(* IEC 61131-3 sources: ATCMcontrol_Engineering/src/Target/ATHW119/Libs/ATCM_Utility, 30 files *)

(* ---- BYTE_SWAP_DWORD.st ---- *)
(*[[
    UserURL= "ATCMfile:BYTE_SWAP_DWORD.htm"
]]*)

(* swaps from big to little endian byte order and vice versa *)

FUNCTION BYTE_SWAP_DWORD : DWORD
VAR_INPUT
    VALUE : DWORD;
END_VAR

inline { STDLIB ( byte_swap_dword ) }

END_FUNCTION

(* ---- BYTE_SWAP_WORD.st ---- *)
(*[[
    UserURL= "ATCMfile:BYTE_SWAP_WORD.htm"
]]*)

(* swaps from big to little endian byte order and vice versa *)

FUNCTION BYTE_SWAP_WORD : WORD
VAR_INPUT
    VALUE : WORD;
END_VAR

inline { STDLIB ( byte_swap_word ) }

END_FUNCTION

(* ---- COPY_BOOL_FROM_BYTE_ARRAY.st ---- *)
(*[[
    UserURL= "ATCMfile:COPY_BOOL_FROM_BYTE_ARRAY.htm"
]]*)

(* returns a value copied from the byte array at the position POS *)

FUNCTION COPY_BOOL_FROM_BYTE_ARRAY : BOOL
VAR_IN_OUT
    POS : DINT;
    BYTES : ARRAY OF BYTE;
END_VAR

inline { STDLIB ( copy_bool_from_byte_array ) }

END_FUNCTION

(* ---- COPY_BOOL_TO_BYTE_ARRAY.st ---- *)
(*[[
    UserURL= "ATCMfile:COPY_BOOL_TO_BYTE_ARRAY.htm"
]]*)

(* copies the value VALUE to the byte array at the position POS *)

FUNCTION COPY_BOOL_TO_BYTE_ARRAY
VAR_INPUT
    VALUE : BOOL;
END_VAR
VAR_IN_OUT
    POS : DINT;
    BYTES : ARRAY OF BYTE;
END_VAR

inline { STDLIB ( copy_bool_to_byte_array ) }

END_FUNCTION

(* ---- COPY_BYTE_FROM_BYTE_ARRAY.st ---- *)
(*[[
    UserURL= "ATCMfile:COPY_BYTE_FROM_BYTE_ARRAY.htm"
]]*)

(* returns a value copied from the byte array BYTES at the position POS *)

FUNCTION COPY_BYTE_FROM_BYTE_ARRAY : BYTE
VAR_IN_OUT
    POS : DINT;
    BYTES : ARRAY OF BYTE;
END_VAR

inline { STDLIB ( copy_byte_from_byte_array ) }

END_FUNCTION

(* ---- COPY_BYTE_TO_BYTE_ARRAY.st ---- *)
(*[[
    UserURL= "ATCMfile:COPY_BYTE_TO_BYTE_ARRAY.htm"
]]*)

(* copies the value VALUE to the byte array BYTES at the position POS *)

FUNCTION COPY_BYTE_TO_BYTE_ARRAY
VAR_INPUT
    VALUE : BYTE;
END_VAR
VAR_IN_OUT
    POS : DINT;
    BYTES : ARRAY OF BYTE;
END_VAR

inline { STDLIB ( copy_byte_to_byte_array ) }

END_FUNCTION

(* ---- COPY_DINT_FROM_BYTE_ARRAY.st ---- *)
(*[[
    UserURL= "ATCMfile:COPY_DINT_FROM_BYTE_ARRAY.htm"
]]*)

(* returns a value copied from the byte array BYTES at the position POS *)

FUNCTION COPY_DINT_FROM_BYTE_ARRAY : DINT
VAR_IN_OUT
    POS : DINT;
    BYTES : ARRAY OF BYTE;
END_VAR

inline { STDLIB ( copy_dint_from_byte_array ) }

END_FUNCTION

(* ---- COPY_DINT_TO_BYTE_ARRAY.st ---- *)
(*[[
    UserURL= "ATCMfile:COPY_DINT_TO_BYTE_ARRAY.htm"
]]*)

(* copies the value VALUE to the byte array BYTES at the position POS *)

FUNCTION COPY_DINT_TO_BYTE_ARRAY
VAR_INPUT
    VALUE : DINT;
END_VAR
VAR_IN_OUT
    POS : DINT;
    BYTES : ARRAY OF BYTE;
END_VAR

inline { STDLIB ( copy_dint_to_byte_array ) }

END_FUNCTION

(* ---- COPY_DWORD_FROM_BYTE_ARRAY.st ---- *)
(*[[
    UserURL= "ATCMfile:COPY_DWORD_FROM_BYTE_ARRAY.htm"
]]*)

(* returns a value copied from the byte array at the position POS *)

FUNCTION COPY_DWORD_FROM_BYTE_ARRAY : DWORD
VAR_IN_OUT
    POS : DINT;
    BYTES : ARRAY OF BYTE;
END_VAR

inline { STDLIB ( copy_dword_from_byte_array ) }

END_FUNCTION

(* ---- COPY_DWORD_TO_BYTE_ARRAY.st ---- *)
(*[[
    UserURL= "ATCMfile:COPY_DWORD_TO_BYTE_ARRAY.htm"
]]*)

(* copies the value VALUE to the byte array at the position POS *)

FUNCTION COPY_DWORD_TO_BYTE_ARRAY
VAR_INPUT
    VALUE : DWORD;
END_VAR
VAR_IN_OUT
    POS : DINT;
    BYTES : ARRAY OF BYTE;
END_VAR

inline { STDLIB ( copy_dword_to_byte_array ) }

END_FUNCTION

(* ---- COPY_INT_FROM_BYTE_ARRAY.st ---- *)
(*[[
    UserURL= "ATCMfile:COPY_INT_FROM_BYTE_ARRAY.htm"
]]*)

(* returns a value copied from the byte string BSTR at the position POS *)

FUNCTION COPY_INT_FROM_BYTE_ARRAY : INT
VAR_IN_OUT
    POS : DINT;
    BYTES : ARRAY OF BYTE;
END_VAR

inline { STDLIB ( copy_int_from_byte_array ) }

END_FUNCTION

(* ---- COPY_INT_TO_BYTE_ARRAY.st ---- *)
(*[[
    UserURL= "ATCMfile:COPY_INT_TO_BYTE_ARRAY.htm"
]]*)

(* copies the value VALUE to the byte array BYTES at the position POS *)
FUNCTION COPY_INT_TO_BYTE_ARRAY
VAR_INPUT
    VALUE : INT;
END_VAR
VAR_IN_OUT
    POS : DINT;
    BYTES : ARRAY OF BYTE;
END_VAR

inline { STDLIB ( copy_int_to_byte_array ) }

END_FUNCTION

(* ---- COPY_LREAL_FROM_BYTE_ARRAY.st ---- *)
(*[[
    UserURL= "ATCMfile:COPY_LREAL_FROM_BYTE_ARRAY.htm"
]]*)

(* returns a value copied from the byte string BSTR at the position POS *)

FUNCTION COPY_LREAL_FROM_BYTE_ARRAY : LREAL
VAR_IN_OUT
    POS : DINT;
    BYTES : ARRAY OF BYTE;
END_VAR

inline { STDLIB ( copy_lreal_from_byte_array ) }

END_FUNCTION

(* ---- COPY_LREAL_TO_BYTE_ARRAY.st ---- *)
(*[[
    UserURL= "ATCMfile:COPY_LREAL_TO_BYTE_ARRAY.htm"
]]*)

(* copies the value VALUE to the byte string BSTR at the position POS *)

FUNCTION COPY_LREAL_TO_BYTE_ARRAY
VAR_INPUT
    VALUE : LREAL;
END_VAR
VAR_IN_OUT
    POS : DINT;
    BYTES : ARRAY OF BYTE;
END_VAR

inline { STDLIB ( copy_lreal_to_byte_array ) }

END_FUNCTION

(* ---- COPY_LWORD_FROM_BYTE_ARRAY.st ---- *)
(*[[
    UserURL= "ATCMfile:COPY_LWORD_FROM_BYTE_ARRAY.htm"
]]*)

(* returns a value copied from the byte string BSTR at the position POS *)

FUNCTION COPY_LWORD_FROM_BYTE_ARRAY : LWORD
VAR_IN_OUT
    POS : DINT;
    BYTES : ARRAY OF BYTE;
END_VAR

inline { STDLIB ( copy_lword_from_byte_array ) }

END_FUNCTION

(* ---- COPY_LWORD_TO_BYTE_ARRAY.st ---- *)
(*[[
    UserURL= "ATCMfile:COPY_LWORD_TO_BYTE_ARRAY.htm"
]]*)

(* copies the value VALUE to the byte string BSTR at the position POS *)

FUNCTION COPY_LWORD_TO_BYTE_ARRAY
VAR_INPUT
    VALUE : LWORD;
END_VAR
VAR_IN_OUT
    POS : DINT;
    BYTES : ARRAY OF BYTE;
END_VAR

inline { STDLIB ( copy_lword_to_byte_array ) }

END_FUNCTION

(* ---- COPY_REAL_FROM_BYTE_ARRAY.st ---- *)
(*[[
    UserURL= "ATCMfile:COPY_LREAL_FROM_BYTE_ARRAY.htm"
]]*)

(* returns a value copied from the byte string BSTR at the position POS *)

FUNCTION COPY_REAL_FROM_BYTE_ARRAY : REAL
VAR_IN_OUT
    POS : DINT;
    BYTES : ARRAY OF BYTE;
END_VAR

inline { STDLIB ( copy_real_from_byte_array ) }

END_FUNCTION

(* ---- COPY_REAL_TO_BYTE_ARRAY.st ---- *)
(*[[
    UserURL= "ATCMfile:COPY_LREAL_TO_BYTE_ARRAY.htm"
]]*)

(* copies the value VALUE to the byte string BSTR at the position POS *)

FUNCTION COPY_REAL_TO_BYTE_ARRAY
VAR_INPUT
    VALUE : REAL;
END_VAR
VAR_IN_OUT
    POS : DINT;
    BYTES : ARRAY OF BYTE;
END_VAR

inline { STDLIB ( copy_real_to_byte_array ) }

END_FUNCTION

(* ---- COPY_STRING_FROM_BYTE_ARRAY.st ---- *)
(*[[
    UserURL= "ATCMfile:COPY_STRING_FROM_BYTE_ARRAY.htm"
]]*)

(* Returns a string copied from the byte array
 * at the position POS containing NUM bytes.
 *)
FUNCTION COPY_STRING_FROM_BYTE_ARRAY : STRING
VAR_IN_OUT
    POS : DINT;
    BYTES : ARRAY OF BYTE;
END_VAR

inline { STDLIB ( copy_string_from_byte_array ) }

END_FUNCTION

(* ---- COPY_STRING_TO_BYTE_ARRAY.st ---- *)
(*[[
    UserURL= "ATCMfile:COPY_STRING_TO_BYTE_ARRAY.htm"
]]*)

(* Copies the value VALUE to the byte array BYTES starting at the position POS.
 *)
FUNCTION COPY_STRING_TO_BYTE_ARRAY
VAR_INPUT
    VALUE : STRING;
END_VAR
VAR_IN_OUT
    POS : DINT;
    BYTES : ARRAY OF BYTE;
END_VAR

inline { STDLIB ( copy_string_to_byte_array ) }

END_FUNCTION

(* ---- COPY_TIME_FROM_BYTE_ARRAY.st ---- *)
(*[[
    UserURL= "ATCMfile:COPY_TIME_FROM_BYTE_ARRAY.htm"
]]*)

(* returns a value copied from the byte array BYTES at the position POS *)

FUNCTION COPY_TIME_FROM_BYTE_ARRAY : TIME
VAR_IN_OUT
    POS : DINT;
    BYTES : ARRAY OF BYTE;
END_VAR

inline { STDLIB ( copy_time_from_byte_array ) }

END_FUNCTION

(* ---- COPY_TIME_TO_BYTE_ARRAY.st ---- *)
(*[[
    UserURL= "ATCMfile:COPY_TIME_TO_BYTE_ARRAY.htm"
]]*)

(* copies the value VALUE to the byte array BYTES at the position POS *)

FUNCTION COPY_TIME_TO_BYTE_ARRAY
VAR_INPUT
    VALUE : TIME;
END_VAR
VAR_IN_OUT
    POS : DINT;
    BYTES : ARRAY OF BYTE;
END_VAR

inline { STDLIB ( copy_time_to_byte_array ) }

END_FUNCTION

(* ---- COPY_WORD_FROM_BYTE_ARRAY.st ---- *)
(*[[
    UserURL= "ATCMfile:COPY_WORD_FROM_BYTE_ARRAY.htm"
]]*)

(* returns a value copied from the byte array BYTES at the position POS *)

FUNCTION COPY_WORD_FROM_BYTE_ARRAY : WORD
VAR_IN_OUT
    POS : DINT;
    BYTES : ARRAY OF BYTE;
END_VAR

inline { STDLIB ( copy_word_from_byte_array ) }

END_FUNCTION

(* ---- COPY_WORD_TO_BYTE_ARRAY.st ---- *)
(*[[
    UserURL= "ATCMfile:COPY_WORD_TO_BYTE_ARRAY.htm"
]]*)

(* copies the value VALUE to the byte array BYTES at the position POS *)

FUNCTION COPY_WORD_TO_BYTE_ARRAY
VAR_INPUT
    VALUE : WORD;
END_VAR
VAR_IN_OUT
    POS : DINT;
    BYTES : ARRAY OF BYTE;
END_VAR

inline { STDLIB ( copy_word_to_byte_array ) }

END_FUNCTION

(* ---- HI_BYTE.st ---- *)
(*[[
    UserURL= "ATCMfile:HI_BYTE.htm"
]]*)

(* extracts the high value BYTE from a WORD *)

FUNCTION HI_BYTE : BYTE
VAR_INPUT
    VALUE : WORD;
END_VAR

inline { STDLIB ( hi_byte ) }

END_FUNCTION

(* ---- HI_WORD.st ---- *)
(*[[
    UserURL= "ATCMfile:HI_WORD.htm"
]]*)

(* extracts the high value WORD from a DWORD *)

FUNCTION HI_WORD : WORD
VAR_INPUT
    VALUE : DWORD;
END_VAR

inline { STDLIB ( hi_word ) }

END_FUNCTION

(* ---- LO_BYTE.st ---- *)
(*[[
    UserURL= "ATCMfile:LO_BYTE.htm"
]]*)

(* extracts the low value BYTE from a WORD *)

FUNCTION LO_BYTE : BYTE
VAR_INPUT
    VALUE : WORD;
END_VAR

inline { STDLIB ( lo_byte ) }

END_FUNCTION

(* ---- LO_WORD.st ---- *)
(*[[
    UserURL= "ATCMfile:LO_WORD.htm"
]]*)

(* extracts the low value WORD from a DWORD *)

FUNCTION LO_WORD : WORD
VAR_INPUT
    VALUE : DWORD;
END_VAR

inline { STDLIB ( lo_word ) }

END_FUNCTION

(* ---- MAKE_DWORD.st ---- *)
(*[[
    UserURL= "ATCMfile:MAKE_DWORD.htm"
]]*)

(* combines two WORDs to a DWORD *)

FUNCTION MAKE_DWORD : DWORD
VAR_INPUT
    LO_WORD : WORD;
    HI_WORD : WORD;
END_VAR

inline { STDLIB ( make_dword ) }

END_FUNCTION

(* ---- MAKE_WORD.st ---- *)
(*[[
    UserURL= "ATCMfile:MAKE_WORD.htm"
]]*)

(* combines two BYTEs to a WORD *)

FUNCTION MAKE_WORD : WORD
VAR_INPUT
    LO_BYTE : BYTE;
    HI_BYTE : BYTE;
END_VAR

inline { STDLIB ( make_word ) }

END_FUNCTION
